(* Logix 5000 project; controller cal1615 1756-L62 rev 20.11; software revision 20.05; part 40 of 82 *)
(* tags used below, declared in another part *)
   FAULT : BOOL;   // Fault AFI
   p01_recipe_active : recipe;   // Active Recipe
   p01r09_pb_global_reset : BOOL;   // System Modes PB: Global Fault Reset
   p01r13_permissive_drives : BOOL;   // System Line Start Sequence Permissive Drives
   p02_dint_from_hmi : hmi_dint;
   p02_real_from_hmi : hmi_real;   // MOP HMI Iface Real from HMI
   p20_ai_lc01 : REAL;   // Letoff Analog Input Line Tension Load Cell Splicer
   p20_di_acc_empty : BOOL;   // Letoff Digital Input Letoff Accumulator Empty Position
   p20_di_lfr_jog_fwd : BOOL;   // Letoff Digital Input PB: Feedroll Jog Forward
   p20_di_lfr_jog_rev : BOOL;   // Letoff Digital Input PB: Feedroll Jog Reverse
   p20_di_lfr_nip_close : BOOL;   // Letoff Digital Input PB: Feedroll Nip Roll Close
   p20_di_loa_active : BOOL;   // Letoff Digital Input Letoff A Active
   p20_di_loa_fwd_dir : BOOL;   // Letoff Digital Inputs PB: Letoff A Jog FWD
   p20_di_lob_fwd_dir : BOOL;   // Letoff Digital Inputs PB: Letoff B Jog FWD
   p20_do_close_nip : BOOL;   // Letoff Digital Output Feedroll Roll Nip Close
   p20_do_enable_lfr_fwd : BOOL;   // Letoff Digital Output Letoff Accumulator Feedroll Forward
   p20_do_enable_lfr_rev : BOOL;   // Letoff Digital Output Letoff Accumulator Feedroll Reverse
   p20_do_engage_lfr_clutch : BOOL;   // Letoff Digital Output Engage Letoff Accumulator Feedroll Clutch
   p20_param_high_ki : REAL;
   p20_param_high_kp : REAL;
   p20_param_high_upd : REAL;
   p20r01 : routine;   // Letoff Main
   p20r09 : routine;   // Letoff Modes
   p20r09_acc_toggle : SYS_Toggle;   // Letoff Modes Accumulator Auto
   p20r09_accumulator_auto : BOOL;   // Letoff Modes Accumulator Auto Mode
   p20r09_letoff_a_active : BOOL;   // Letoff Modes Letoff A Active
   p20r09_timer_fault : TIMER[4];   // Letoff Modes Fault Delay
   p20r09_timer_warning : TIMER[4];   // Letoff Modes Warning Delay
   p20r10 : routine;   // Letoff Letoff Tension Control
   p20r10_param_acc_full_psn : REAL;
   p20r10_param_fill_gain : REAL;
   p20r10_param_normal_gain : REAL;
   p20r10_param_psn_gain : REAL;   // Letoff Letoff Tension Control Tension Gain
   p20r10_pid_psn : PID;   // Letoff Letoff Position Control PID
   p20r10_pid_psn_cv : REAL;
   p20r10_pid_psn_pv : REAL;   // Letoff Letoff Positon Control PID Process Value
   p20r10_pid_tens : PID;   // Letoff Letoff Speed Control Tension PID
   p20r10_pid_tens_cv : REAL;   // Letoff Letoff Speed Control Control Value CV
   p20r10_pid_tens_pv : REAL;   // Letoff Letoff Tension Control PID Process Value
   p20r10_run_permissive : BOOL;   // Letoff Letoff Tension Control Run Permissive
   p20r10_speed_offset : REAL;   // Letoff Letoff Speed Control Speed Offset
   p20r10_speed_offset_psn : REAL;   // Letoff Letoff Speed Control Position PID Speed Offset
   p20r10_speed_offset_tens : REAL;   // Letoff Letoff Speed Control Tension PID Speed Offset
   p20r10_tension_request : BOOL;   // Letoff Letoff Tension Control Tension Control Request
   p20r10_timer : TIMER[2];   // Letoff Letoff Tension Control PID Condition
   p20r10_timer_fault : TIMER[4];   // Letoff Fault Delay
   p20r10_timer_warning : TIMER[4];   // Letoff Warning Delay
   p20r11 : routine;   // Letoff Feedroll
   p20r11_manual_open_nip : BOOL;   // Letoff Feedroll Request Manual Open Nip
   p20r11_nip_close_dwell : TIMER;
   p20r11_permissive_jog : BOOL;   // Letoff Feedroll Permissive Jog
   p20r11_permissive_run : BOOL;   // Letoff Feedroll Permissive Run
   p20r11_request_close_nip : BOOL;   // Letoff Feedroll Request Close Feedroll Nip Roll
   p20r11_request_jog_fwd : BOOL;   // Letoff Feedroll Request Jog Forward
   p20r11_request_jog_rev : BOOL;   // Letoff Feedroll Request Jog Reverse
   p20r11_timer_clutch_off : TIMER;   // Letoff Feedroll Clutch Off Delay
   p20r11_timer_clutch_on : TIMER;   // Letoff Feedroll Clutch On Delay
   p20r11_timer_fault : TIMER[4];   // Letoff Feedroll Fault Delay
   p20r11_timer_warning : TIMER[4];   // Letoff Feedroll Warning Delay
   p20r13_ai_acc_pct : REAL;   // Letoff Accumulator Pct Full
   p20r13_state : DINT;   // Letoff Accumulator State
   p20r15_request_tension : BOOL;   // Letoff Letoff A VFD Request Tension
   p20r15_request_thread_fwd : BOOL;
   p20r15_request_thread_rev : BOOL;
   p20r16_request_tension : BOOL;   // Letoff Letoff B VFD Request Tension
   p20r16_request_thread_fwd : BOOL;
   p20r16_request_thread_rev : BOOL;
   p21_di_open_splice_platen : BOOL;   // Splice Press Digital Input Open Platen
   p21r10_state : DINT;   // Splice Press Sequence State
   p30r10_state : DINT;   // Splice Press Sequence State
(* P20_Letoff, continued *)

ROUTINE R09_Modes   (* ladder *)
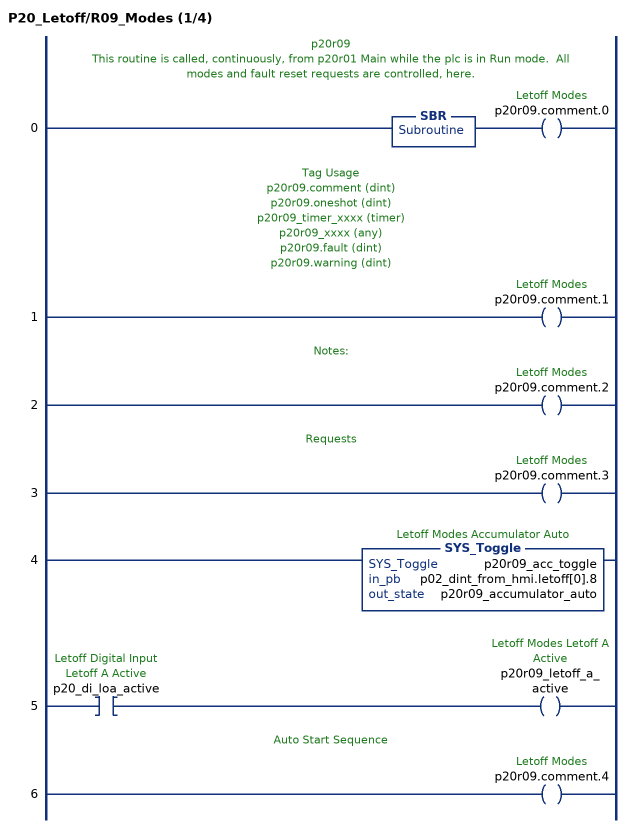
   // p20r09
   // This routine is called, continuously, from p20r01 Main while the plc is in Run mode.  All modes and fault reset requests are controlled, here.
   0: SBR()OTE(p20r09.comment.0);
   // Tag Usage
   // p20r09.comment (dint)
   // p20r09.oneshot (dint)
   // p20r09_timer_xxxx (timer)
   // p20r09_xxxx (any)
   // p20r09.fault (dint)
   // p20r09.warning (dint)
   1: OTE(p20r09.comment.1);
   // Notes:
   2: OTE(p20r09.comment.2);
   // Requests
   3: OTE(p20r09.comment.3);
   4: SYS_Toggle(p20r09_acc_toggle,p02_dint_from_hmi.letoff[0].8,p20r09_accumulator_auto);
   5: XIC(p20_di_loa_active)OTE(p20r09_letoff_a_active);
   // Auto Start Sequence
   6: OTE(p20r09.comment.4);
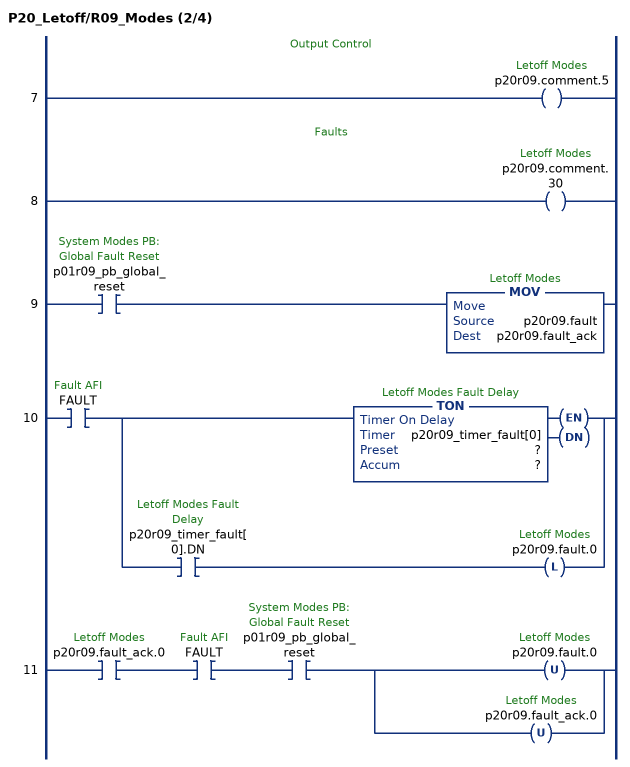
   // Output Control
   7: OTE(p20r09.comment.5);
   // Faults
   8: OTE(p20r09.comment.30);
   9: XIC(p01r09_pb_global_reset)MOV(p20r09.fault,p20r09.fault_ack);
   10: XIC(FAULT)[TON(p20r09_timer_fault[0],?,?) ,XIC(p20r09_timer_fault[0].DN) OTL(p20r09.fault.0) ];
   11: XIC(p20r09.fault_ack.0)XIC(FAULT)XIC(p01r09_pb_global_reset)[OTU(p20r09.fault.0) ,OTU(p20r09.fault_ack.0) ];
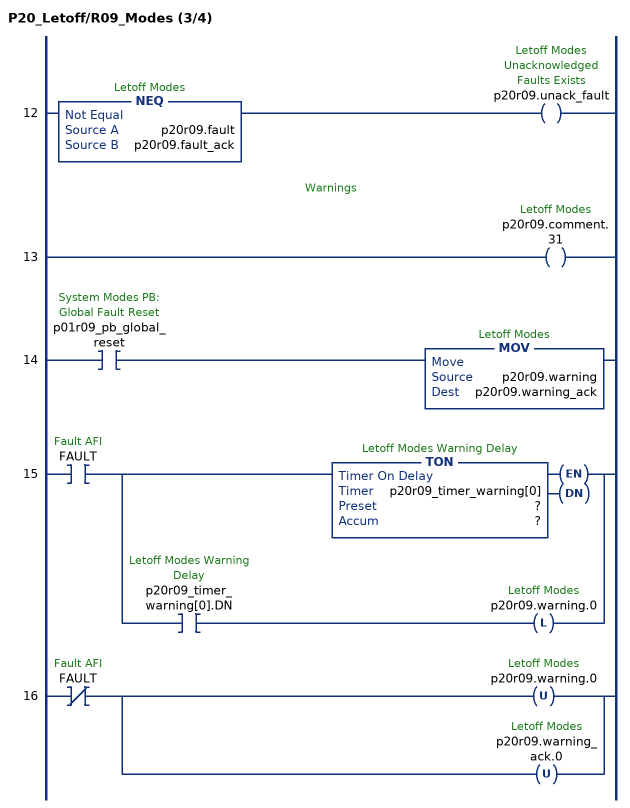
   12: NEQ(p20r09.fault,p20r09.fault_ack)OTE(p20r09.unack_fault);
   // Warnings
   13: OTE(p20r09.comment.31);
   14: XIC(p01r09_pb_global_reset)MOV(p20r09.warning,p20r09.warning_ack);
   15: XIC(FAULT)[TON(p20r09_timer_warning[0],?,?) ,XIC(p20r09_timer_warning[0].DN) OTL(p20r09.warning.0) ];
   16: XIO(FAULT)[OTU(p20r09.warning.0) ,OTU(p20r09.warning_ack.0) ];
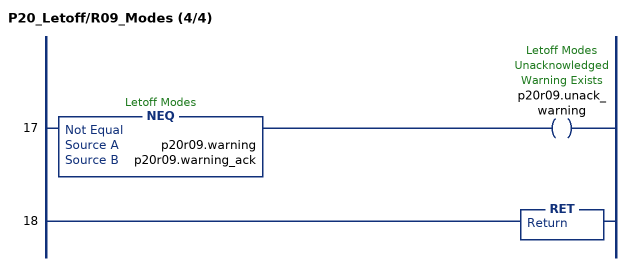
   17: NEQ(p20r09.warning,p20r09.warning_ack)OTE(p20r09.unack_warning);
   18: RET();
END_ROUTINE

ROUTINE R10_Letoff_Speed_Control   (* ladder *)
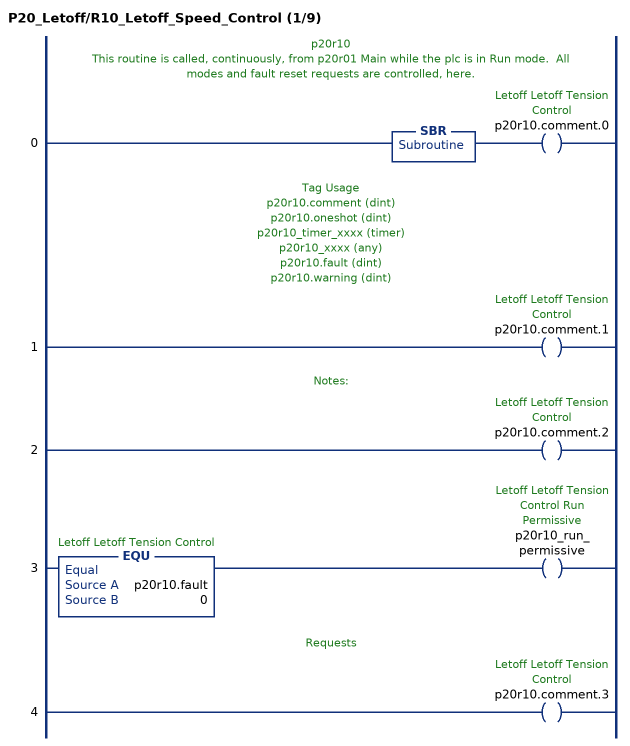
   // p20r10
   // This routine is called, continuously, from p20r01 Main while the plc is in Run mode.  All modes and fault reset requests are controlled, here.
   0: SBR()OTE(p20r10.comment.0);
   // Tag Usage
   // p20r10.comment (dint)
   // p20r10.oneshot (dint)
   // p20r10_timer_xxxx (timer)
   // p20r10_xxxx (any)
   // p20r10.fault (dint)
   // p20r10.warning (dint)
   1: OTE(p20r10.comment.1);
   // Notes:
   2: OTE(p20r10.comment.2);
   3: EQU(p20r10.fault,0)OTE(p20r10_run_permissive);
   // Requests
   4: OTE(p20r10.comment.3);
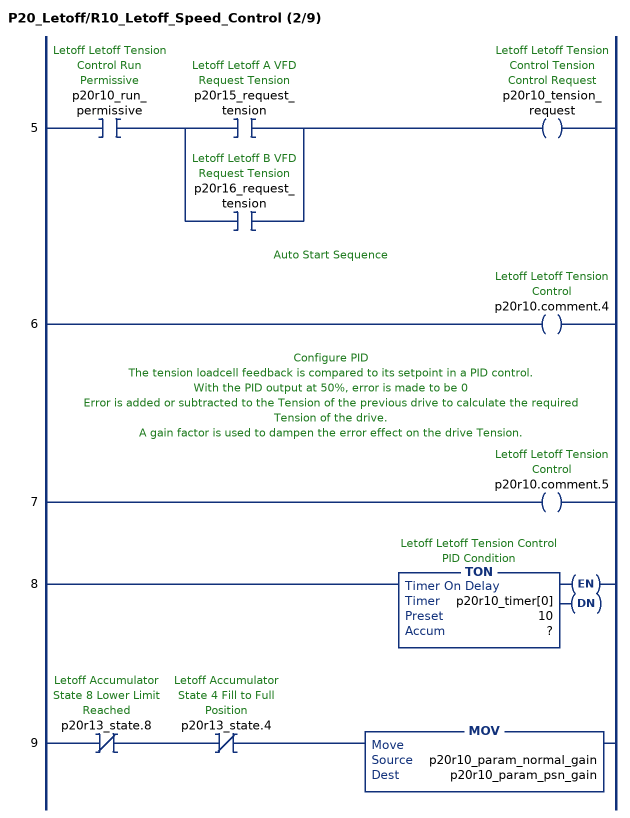
   5: XIC(p20r10_run_permissive)[XIC(p20r15_request_tension) ,XIC(p20r16_request_tension) ]OTE(p20r10_tension_request);
   // Auto Start Sequence
   6: OTE(p20r10.comment.4);
   // Configure PID
   // The tension loadcell feedback is compared to its setpoint in a PID control.
   // With the PID output at 50%, error is made to be 0
   // Error is added or subtracted to the Tension of the previous drive to calculate the required Tension of the drive.
   // A gain factor is used to dampen the error effect on the drive Tension.
   7: OTE(p20r10.comment.5);
   8: TON(p20r10_timer[0],?,?);
   9: XIO(p20r13_state.8)XIO(p20r13_state.4)MOV(p20r10_param_normal_gain,p20r10_param_psn_gain);
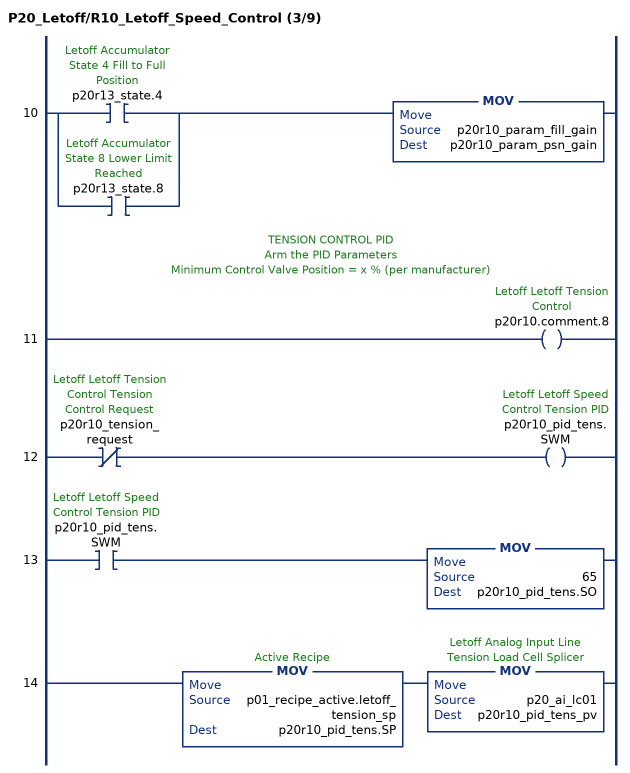
   10: [XIC(p20r13_state.4) ,XIC(p20r13_state.8) ]MOV(p20r10_param_fill_gain,p20r10_param_psn_gain);
   // TENSION CONTROL PID
   // Arm the PID Parameters
   // Minimum Control Valve Position = x % (per manufacturer)
   11: OTE(p20r10.comment.8);
   12: XIO(p20r10_tension_request)OTE(p20r10_pid_tens.SWM);
   13: XIC(p20r10_pid_tens.SWM)MOV(65,p20r10_pid_tens.SO);
   14: MOV(p01_recipe_active.letoff_tension_sp,p20r10_pid_tens.SP)MOV(p20_ai_lc01,p20r10_pid_tens_pv);
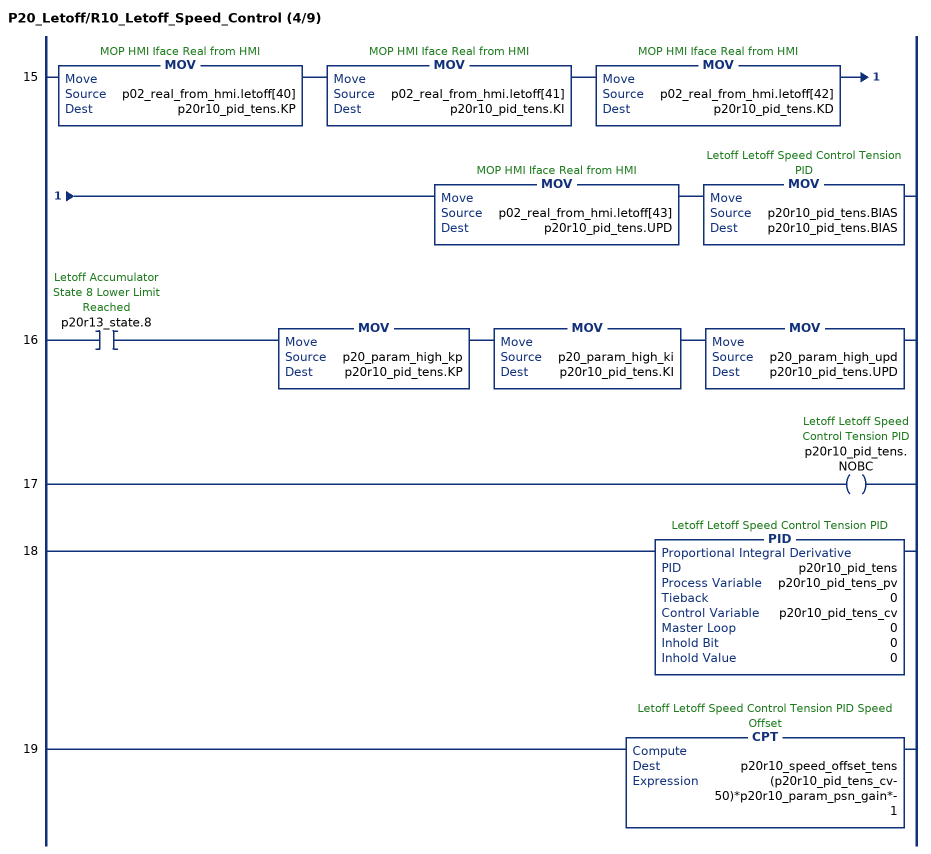
   15: MOV(p02_real_from_hmi.letoff[40],p20r10_pid_tens.KP)MOV(p02_real_from_hmi.letoff[41],p20r10_pid_tens.KI)MOV(p02_real_from_hmi.letoff[42],p20r10_pid_tens.KD)MOV(p02_real_from_hmi.letoff[43],p20r10_pid_tens.UPD)MOV(p20r10_pid_tens.BIAS,p20r10_pid_tens.BIAS);
   16: XIC(p20r13_state.8)MOV(p20_param_high_kp,p20r10_pid_tens.KP)MOV(p20_param_high_ki,p20r10_pid_tens.KI)MOV(p20_param_high_upd,p20r10_pid_tens.UPD);
   17: OTE(p20r10_pid_tens.NOBC);
   18: PID(p20r10_pid_tens,p20r10_pid_tens_pv,0,p20r10_pid_tens_cv,0,0,0);
   19: CPT(p20r10_speed_offset_tens,(p20r10_pid_tens_cv-50)*p20r10_param_psn_gain*-1);
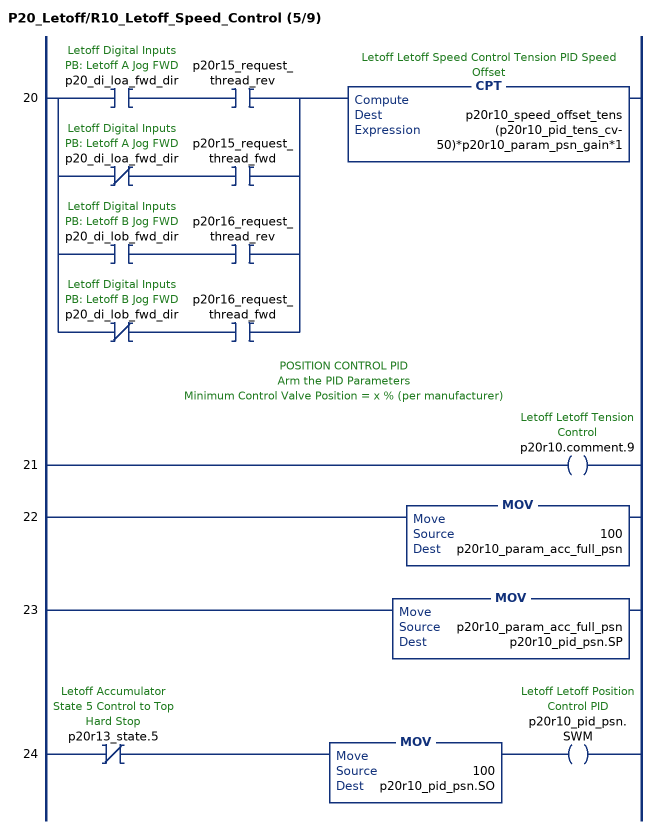
   20: [XIC(p20_di_loa_fwd_dir) XIC(p20r15_request_thread_rev) ,XIO(p20_di_loa_fwd_dir) XIC(p20r15_request_thread_fwd) ,XIC(p20_di_lob_fwd_dir) XIC(p20r16_request_thread_rev) ,XIO(p20_di_lob_fwd_dir) XIC(p20r16_request_thread_fwd) ]CPT(p20r10_speed_offset_tens,(p20r10_pid_tens_cv-50)*p20r10_param_psn_gain*1);
   // POSITION CONTROL PID
   // Arm the PID Parameters
   // Minimum Control Valve Position = x % (per manufacturer)
   21: OTE(p20r10.comment.9);
   22: MOV(100,p20r10_param_acc_full_psn);
   23: MOV(p20r10_param_acc_full_psn,p20r10_pid_psn.SP);
   24: XIO(p20r13_state.5)MOV(100,p20r10_pid_psn.SO)OTE(p20r10_pid_psn.SWM);
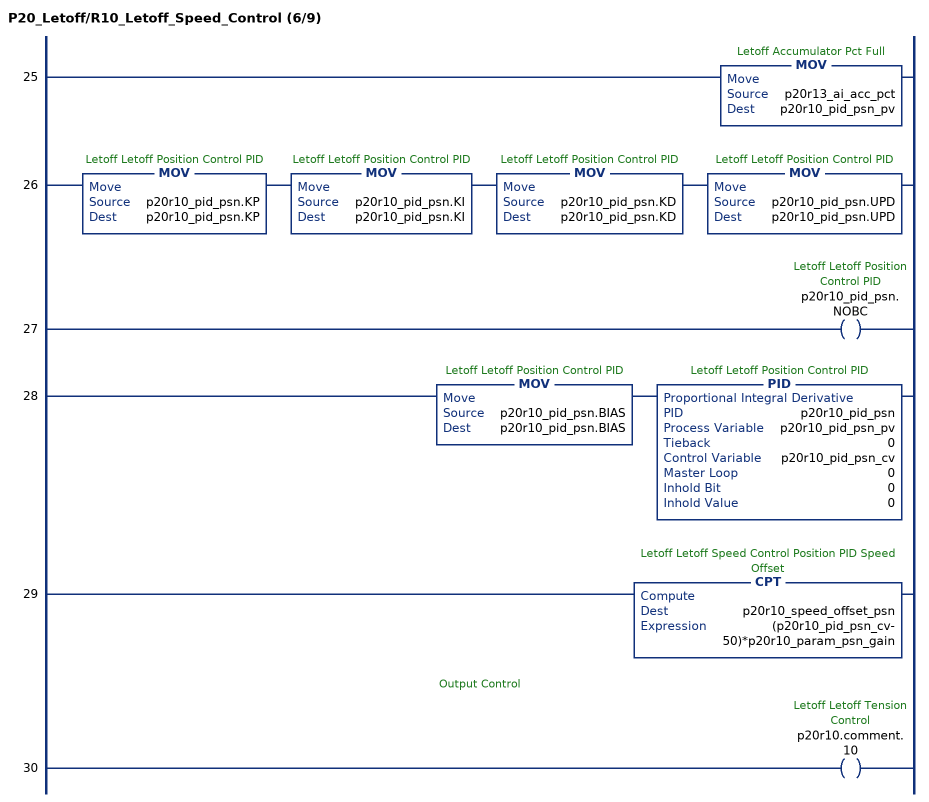
   25: MOV(p20r13_ai_acc_pct,p20r10_pid_psn_pv);
   26: MOV(p20r10_pid_psn.KP,p20r10_pid_psn.KP)MOV(p20r10_pid_psn.KI,p20r10_pid_psn.KI)MOV(p20r10_pid_psn.KD,p20r10_pid_psn.KD)MOV(p20r10_pid_psn.UPD,p20r10_pid_psn.UPD);
   27: OTE(p20r10_pid_psn.NOBC);
   28: MOV(p20r10_pid_psn.BIAS,p20r10_pid_psn.BIAS)PID(p20r10_pid_psn,p20r10_pid_psn_pv,0,p20r10_pid_psn_cv,0,0,0);
   29: CPT(p20r10_speed_offset_psn,(p20r10_pid_psn_cv-50)*p20r10_param_psn_gain);
   // Output Control
   30: OTE(p20r10.comment.10);
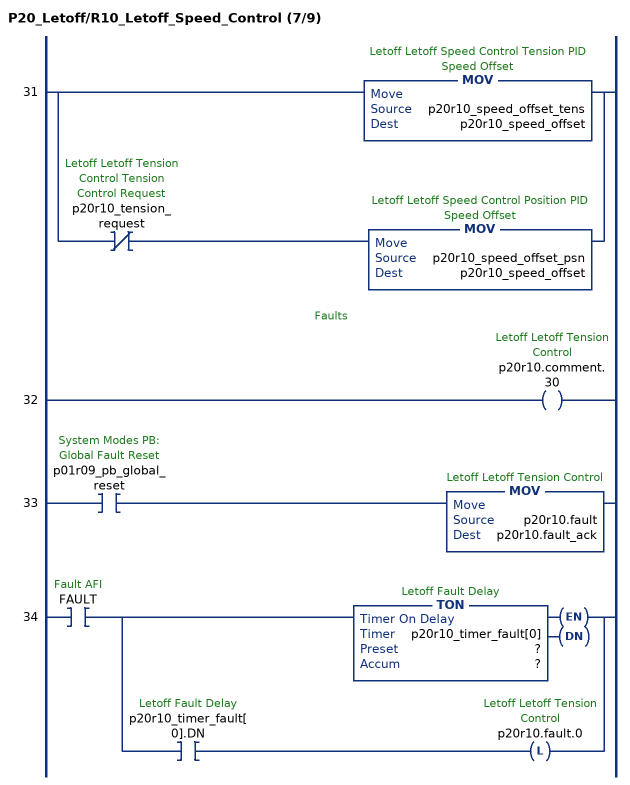
   31: [MOV(p20r10_speed_offset_tens,p20r10_speed_offset) ,XIO(p20r10_tension_request) MOV(p20r10_speed_offset_psn,p20r10_speed_offset) ];
   // Faults
   32: OTE(p20r10.comment.30);
   33: XIC(p01r09_pb_global_reset)MOV(p20r10.fault,p20r10.fault_ack);
   34: XIC(FAULT)[TON(p20r10_timer_fault[0],?,?) ,XIC(p20r10_timer_fault[0].DN) OTL(p20r10.fault.0) ];
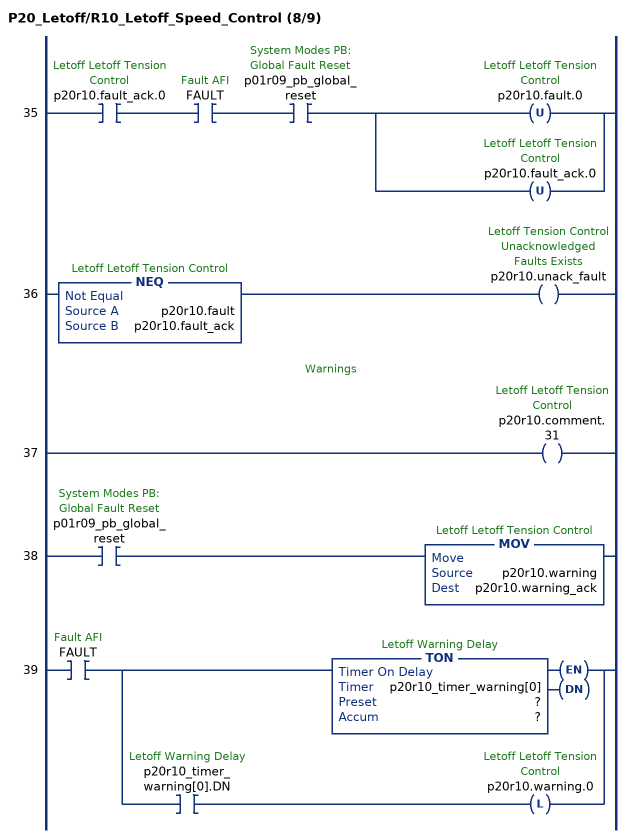
   35: XIC(p20r10.fault_ack.0)XIC(FAULT)XIC(p01r09_pb_global_reset)[OTU(p20r10.fault.0) ,OTU(p20r10.fault_ack.0) ];
   36: NEQ(p20r10.fault,p20r10.fault_ack)OTE(p20r10.unack_fault);
   // Warnings
   37: OTE(p20r10.comment.31);
   38: XIC(p01r09_pb_global_reset)MOV(p20r10.warning,p20r10.warning_ack);
   39: XIC(FAULT)[TON(p20r10_timer_warning[0],?,?) ,XIC(p20r10_timer_warning[0].DN) OTL(p20r10.warning.0) ];
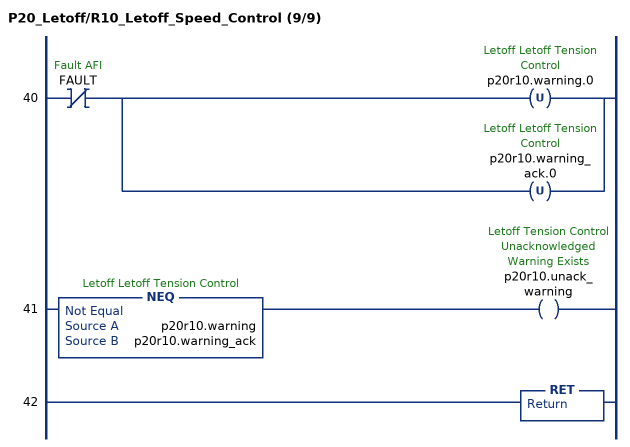
   40: XIO(FAULT)[OTU(p20r10.warning.0) ,OTU(p20r10.warning_ack.0) ];
   41: NEQ(p20r10.warning,p20r10.warning_ack)OTE(p20r10.unack_warning);
   42: RET();
END_ROUTINE

ROUTINE R11_Feedroll   (* ladder *)
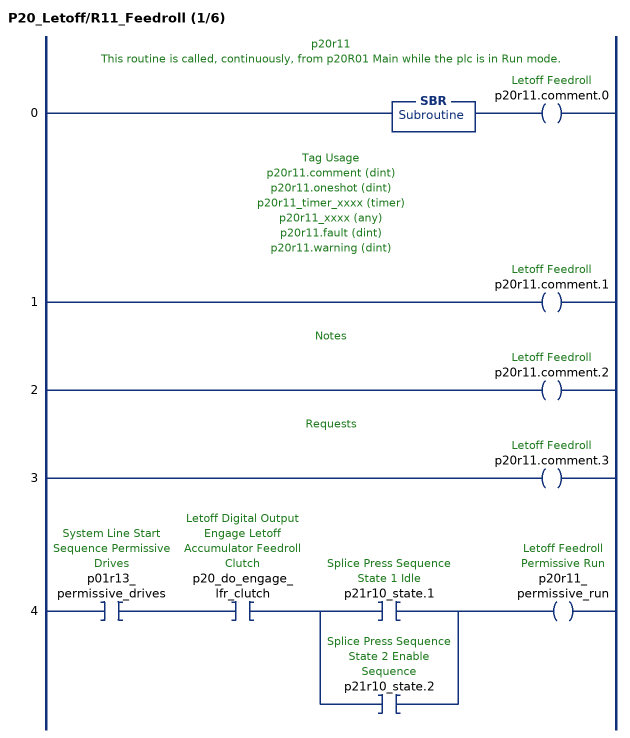
   // p20r11
   // This routine is called, continuously, from p20R01 Main while the plc is in Run mode.
   0: SBR()OTE(p20r11.comment.0);
   // Tag Usage
   // p20r11.comment (dint)
   // p20r11.oneshot (dint)
   // p20r11_timer_xxxx (timer)
   // p20r11_xxxx (any)
   // p20r11.fault (dint)
   // p20r11.warning (dint)
   1: OTE(p20r11.comment.1);
   // Notes
   2: OTE(p20r11.comment.2);
   // Requests
   3: OTE(p20r11.comment.3);
   4: XIC(p01r13_permissive_drives)XIC(p20_do_engage_lfr_clutch)[XIC(p21r10_state.1) ,XIC(p21r10_state.2) ]OTE(p20r11_permissive_run);
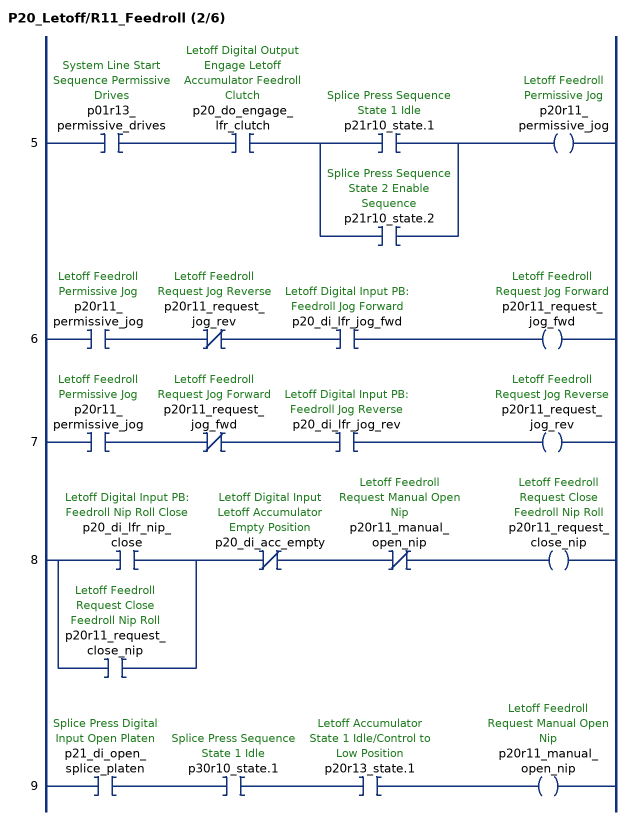
   5: XIC(p01r13_permissive_drives)XIC(p20_do_engage_lfr_clutch)[XIC(p21r10_state.1) ,XIC(p21r10_state.2) ]OTE(p20r11_permissive_jog);
   6: XIC(p20r11_permissive_jog)XIO(p20r11_request_jog_rev)XIC(p20_di_lfr_jog_fwd)OTE(p20r11_request_jog_fwd);
   7: XIC(p20r11_permissive_jog)XIO(p20r11_request_jog_fwd)XIC(p20_di_lfr_jog_rev)OTE(p20r11_request_jog_rev);
   8: [XIC(p20_di_lfr_nip_close) ,XIC(p20r11_request_close_nip) ]XIO(p20_di_acc_empty)XIO(p20r11_manual_open_nip)OTE(p20r11_request_close_nip);
   9: XIC(p21_di_open_splice_platen)XIC(p30r10_state.1)XIC(p20r13_state.1)OTE(p20r11_manual_open_nip);
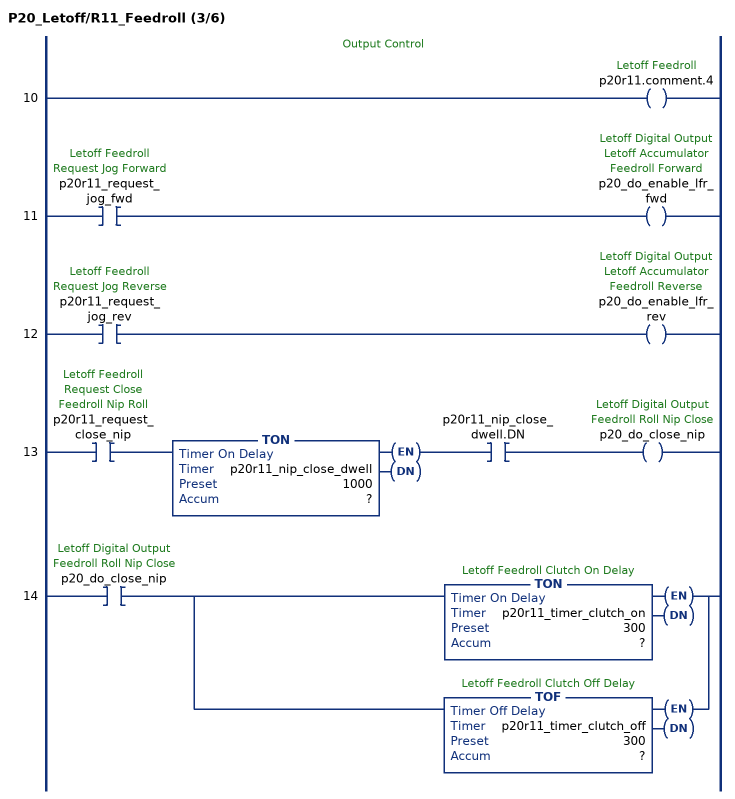
   // Output Control
   10: OTE(p20r11.comment.4);
   11: XIC(p20r11_request_jog_fwd)OTE(p20_do_enable_lfr_fwd);
   12: XIC(p20r11_request_jog_rev)OTE(p20_do_enable_lfr_rev);
   13: XIC(p20r11_request_close_nip)TON(p20r11_nip_close_dwell,?,?)XIC(p20r11_nip_close_dwell.DN)OTE(p20_do_close_nip);
   14: XIC(p20_do_close_nip)[TON(p20r11_timer_clutch_on,?,?) ,TOF(p20r11_timer_clutch_off,?,?) ];
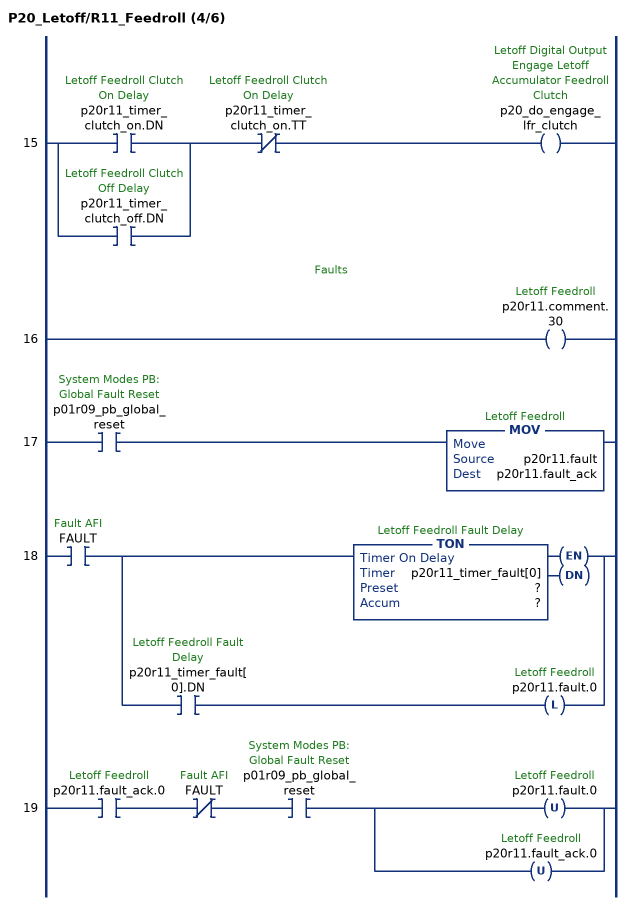
   15: [XIC(p20r11_timer_clutch_on.DN) ,XIC(p20r11_timer_clutch_off.DN) ]XIO(p20r11_timer_clutch_on.TT)OTE(p20_do_engage_lfr_clutch);
   // Faults
   16: OTE(p20r11.comment.30);
   17: XIC(p01r09_pb_global_reset)MOV(p20r11.fault,p20r11.fault_ack);
   18: XIC(FAULT)[TON(p20r11_timer_fault[0],?,?) ,XIC(p20r11_timer_fault[0].DN) OTL(p20r11.fault.0) ];
   19: XIC(p20r11.fault_ack.0)XIO(FAULT)XIC(p01r09_pb_global_reset)[OTU(p20r11.fault.0) ,OTU(p20r11.fault_ack.0) ];
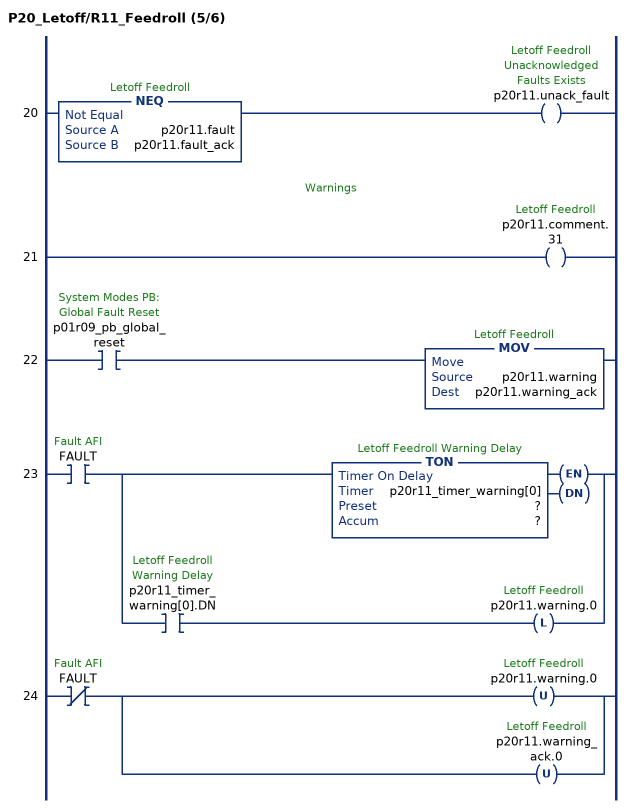
   20: NEQ(p20r11.fault,p20r11.fault_ack)OTE(p20r11.unack_fault);
   // Warnings
   21: OTE(p20r11.comment.31);
   22: XIC(p01r09_pb_global_reset)MOV(p20r11.warning,p20r11.warning_ack);
   23: XIC(FAULT)[TON(p20r11_timer_warning[0],?,?) ,XIC(p20r11_timer_warning[0].DN) OTL(p20r11.warning.0) ];
   24: XIO(FAULT)[OTU(p20r11.warning.0) ,OTU(p20r11.warning_ack.0) ];
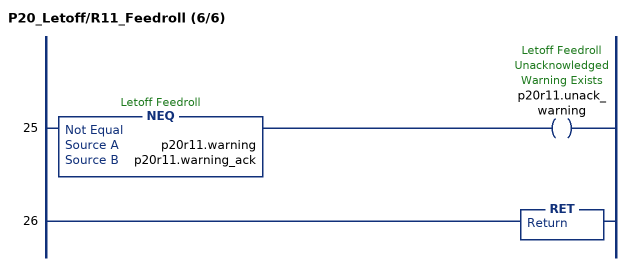
   25: NEQ(p20r11.warning,p20r11.warning_ack)OTE(p20r11.unack_warning);
   26: RET();
END_ROUTINE
